KUKA KRL program: 45degree_axel_test.src

&ACCESS RVP
&REL 1
&PARAM TEMPLATE = C:\KRC\Roboter\Template\vorgabe
&PARAM EDITMASK = *
DEF Prog3 ( )
EXT BAS (BAS_COMMAND :IN,REAL :IN )


; GLOBAL INTERRUPT DECL 3 WHEN $STOPMESS==TRUE DO IR_STOPM ( )
; INTERRUPT ON 3

;FOLD Initialise and set default speed
BAS (#INITMOV,0)
BAS (#VEL_PTP,100)
BAS (#ACC_PTP,20)
$VEL.CP=0.2
BAS (#TOOL,0)
BAS (#BASE,0)
;ENDFOLD

;;FOLD STARTPOS
;$BWDSTART = FALSE
;PDAT_ACT = PDEFAULT
;BAS(#PTP_DAT)
;FDAT_ACT = {TOOL_NO 0,BASE_NO 0,IPO_FRAME #BASE}
;BAS(#FRAMES)
;;ENDFOLD

$ADVANCE = 5

;FOLD ---- Quickly skip BCO ----
; PTP $AXIS_ACT
;ENDFOLD

;FOLD ---- GO HOME ----
; PTP {A1 0.000, A2 -90.000, A3 90.000, A4 0.000, A5 0.000, A6 0.000, E1 0, E2 0, E3 0, E4 0, E5 0, E6 0}
;ENDFOLD


; Program generated by RoboDK v5.9.4 for KUKA KR 90 R2700 pro on 12/01/2026 08:53:20
; Using nominal kinematics.
; ---- Setting reference (Base) ----
$BASE = {FRAME: X 0.000,Y 0.000,Z 0.000,A 0.000,B 0.000,C 0.000}
; BASE_DATA[1] = {FRAME: X 0.000,Y 0.000,Z 0.000,A 0.000,B 0.000,C 0.000}
; $BASE = BASE_DATA[1]
; --------------------------
PTP {A1 0.00000,A2 0.00000,A3 0.00000,A4 0.00000,A5 0.00000,A6 0.00000}
PTP {A1 45.0, A2 0.0, A3 0.0, A4 0.0, A5 0.0, A6 0.0}
PTP {A1 -45.0, A2 0.0, A3 0.0, A4 0.0, A5 0.0, A6 0.0}
PTP {A1 0.00000,A2 0.00000,A3 0.00000,A4 0.00000,A5 0.00000,A6 0.00000}
PTP {A1 0.00000, A2 45.00000, A3 0.00000, A4 0.00000, A5 0.00000, A6 0.00000}
PTP {A1 0.00000, A2 -45.00000, A3 0.00000, A4 0.00000, A5 0.00000, A6 0.00000}
PTP {A1 0.00000,A2 0.00000,A3 0.00000,A4 0.00000,A5 0.00000,A6 0.00000}
PTP {A1 0.00000, A2 0.00000, A3 45.00000, A4 0.00000, A5 0.00000, A6 0.00000}
PTP {A1 0.00000, A2 0.00000, A3 -45.00000, A4 0.00000, A5 0.00000, A6 0.00000}
PTP {A1 0.00000,A2 0.00000,A3 0.00000,A4 0.00000,A5 0.00000,A6 0.00000}
PTP {A1 0.00000, A2 0.00000, A3 0.00000, A4 45.00000, A5 0.00000, A6 0.00000}
PTP {A1 0.00000, A2 0.00000, A3 0.00000, A4 -45.00000, A5 0.00000, A6 0.00000}
PTP {A1 0.00000,A2 0.00000,A3 0.00000,A4 0.00000,A5 0.00000,A6 0.00000}
PTP {A1 0.00000, A2 0.00000, A3 0.00000, A4 0.00000, A5 45.00000, A6 0.00000}
PTP {A1 0.00000, A2 0.00000, A3 0.00000, A4 0.00000, A5 -45.00000, A6 0.00000}
PTP {A1 0.00000,A2 0.00000,A3 0.00000,A4 0.00000,A5 0.00000,A6 0.00000}
PTP {A1 0.00000, A2 0.00000, A3 0.00000, A4 0.00000, A5 0.00000, A6 45.00000}
PTP {A1 0.00000, A2 0.00000, A3 0.00000, A4 0.00000, A5 0.00000, A6 -45.00000}
PTP {A1 0.00000,A2 0.00000,A3 0.00000,A4 0.00000,A5 0.00000,A6 0.00000}
END
